/// Supervision function block - system watchdog
PROGRAM INTERNAL P_Supervision
VAR_IN_OUT
	/// Safets IOs
	stIO_Cabinet		: ST_ControlCabinetIO;
		
	/// Logger
	nLogger				: I_Logger;
END_VAR
VAR_INPUT
END_VAR
VAR_OUTPUT
	bError				: BOOL;	
	bWarning			: BOOL;
	
	bCycleStop			: BOOL;
	bFastStop			: BOOL;
END_VAR
VAR
	/// event handler
	IEvent			: I_EventHandler;
	
	/// Hardware diag FB
	fbDiagEtherCAT	: FB_DiagEtherCAT;
	
	/// private var's
	aa									: INT;	
	rTrigMachineStop_Cycle				: R_TRIG;
	rTrigMachineStop_Fast				: R_TRIG;
	tonRstStillstw						: TON;
END_VAR

/// 
/// supervision function block of the project
/// 

// reset

// run supervision (ES, Safety signals, IO-errors, etc.)

// HW diagnostics
M_EcSupervision();
M_ControlCabinet_A01();

// task cycle time exceeded
IF Statics.stPlcSystemInfo.stPlcTaskSystemInfo.CycleTimeExceeded THEN
	IEvent.Select(TC_Events.SystemEventClass.ErrorEvent)
		  .ArgSetWString(stTextListGlobal.stText_System.stText_CycletimeExceeded.wsName)
		  .Raise();	
END_IF


//-------------------------------------------------------------------------------------------------------------

IF HMI.stHmi.stIn.stMain.stButton_Start.bClick AND NOT stGlobalModuleInfo.bStation_All_Auto AND P_Safety.OpMode_Auto THEN
	IEvent.Select(TC_Events.SystemEventClass.InfoEvent)
		  .ArgSetString('Start Auto nicht moeglich -> Station nicht in Betriebsart Auto')
		  .Raise();
END_IF


//-------------------------------------------------------------------------------------------------------------

IF HMI.stHmi.stIn.stMain.stButton_Start.bClick AND NOT P_Safety.OpMode_Auto THEN
	IEvent.Select(TC_Events.SystemEventClass.InfoEvent)
		  .ArgSetString('Start Auto nicht moeglich -> Schlüsselschalter nicht auf Auto')
		  .Raise();
END_IF


//ToDo: stop / fast stop on alarm trigger
//rTrigMachineStop_Cycle(CLK := Services.fbNotiHandler.stNotificationData.eAlarmStopMode = E_EventReaction.CycleStop, Q => bCycleStop);
//rTrigMachineStop_Fast(CLK := Services.fbNotiHandler.stNotificationData.eAlarmStopMode = E_EventReaction.Stop, Q => bFastStop);

/// System error level
{attribute 'monitoring' := 'call'}
PROPERTY Error : BOOL
GET // INTERNAL
Error := bError;
END_GET
END_PROPERTY

METHOD PRIVATE M_ControlCabinet_A01 : BOOL
VAR_INPUT
END_VAR
// EC-Error
IF IO.stControlCabinetIO.stIn.IarrEcStates[E_EtherCatBox.eEtherCatBox_ControlCabinet] <> 8 THEN
	IEvent.Select(TC_Events.EtherCatEventClass.ErrorEvent)
		  .ArgSetString('EtherCatBox Control Cabinet | EC State Error')
		  .Raise();
ELSIF IO.stControlCabinetIO.stIn.IarrEcStates[E_EtherCatBox.eEtherCatBox_Oven_A] <> 8 THEN
	IEvent.Select(TC_Events.EtherCatEventClass.ErrorEvent)
		  .ArgSetString('EtherCatBox Oven A | EC State Error')
		  .Raise();
ELSIF IO.stControlCabinetIO.stIn.IarrEcStates[E_EtherCatBox.eEtherCatBox_Oven_B] <> 8 THEN
	IEvent.Select(TC_Events.EtherCatEventClass.ErrorEvent)
		  .ArgSetString('EtherCatBox Oven B | EC State Error')
		  .Raise();
ELSIF IO.stControlCabinetIO.stIn.IarrEcStates[E_EtherCatBox.eEtherCatBox_Storage] <> 8 THEN
	IEvent.Select(TC_Events.EtherCatEventClass.ErrorEvent)
		  .ArgSetString('EtherCatBox Storage | EC State Error')
		  .Raise();
END_IF
			  
(*	24V-Versorgung Netzgerät 1 Schutzschalter	
ELSIF NOT IO.stControlCabinetIO.stIn.stA01.b24V_NetzSchutz1Ok THEN
	IEvent.Select(TC_Events.HardwareEventClass.ErrorEvent)
			  .ArgSetString('=A01.G10-1QA1 | 24V-Versorgung Netzgerät 1 Schutzschalter NOK')
			  .Raise();
END_IF
*)
END_METHOD

METHOD PRIVATE M_EcSupervision : BOOL
VAR_INPUT
END_VAR
VAR_INST

END_VAR

// automatic EC supervision
fbDiagEtherCAT();

(*
//IarrEcState
// Diag EC Boxes for fast reaction				
IF (stIO_Cabinet.stIn.IarrEcStates[1] <> 8) THEN
	bError:=TRUE;
	fbNotiHandler.M_SetNotificationEx(F_CreateDynText("403",403),
									stTextListGlobal.stText_NG_Hardware, 
									stTextListGlobal.stText_EtherCatBox_Error, "++M1+E2-57CO1 (CU1128)", stTextListGlobal.stText_EtherCatBox_OP_Error, 
									E_AlarmPriority.Error, E_NotificationMode.eNotificationMode_Reset);	
END_IF
IF (stIO_Cabinet.stIn.IarrEcStates[2] <> 8) THEN
	bError:=TRUE;
	fbNotiHandler.M_SetNotificationEx(F_CreateDynText("404",404),
									stTextListGlobal.stText_NG_Hardware, 
									stTextListGlobal.stText_EtherCatBox_Error, "++M1+E2-57CO1 (CU1128-B)", stTextListGlobal.stText_EtherCatBox_OP_Error, 
									E_AlarmPriority.Error, E_NotificationMode.eNotificationMode_Reset);	
END_IF
IF (stIO_Cabinet.stIn.IarrEcStates[3] <> 8) THEN
	bError:=TRUE;
	fbNotiHandler.M_SetNotificationEx(F_CreateDynText("405",405),
									stTextListGlobal.stText_NG_Hardware, 
									stTextListGlobal.stText_EtherCatBox_Error, "++M1+E2-57CO1 (CU1128-C)", stTextListGlobal.stText_EtherCatBox_OP_Error, 
									E_AlarmPriority.Error, E_NotificationMode.eNotificationMode_Reset);	
END_IF
IF (stIO_Cabinet.stIn.IarrEcStates[4] <> 8) THEN
	bError:=TRUE;
	fbNotiHandler.M_SetNotificationEx(F_CreateDynText("406",406),
									stTextListGlobal.stText_NG_Hardware, 
									stTextListGlobal.stText_EtherCatBox_Error, "++M1+E2-62BC1 (EK1100)", stTextListGlobal.stText_EtherCatBox_OP_Error, 
									E_AlarmPriority.Error, E_NotificationMode.eNotificationMode_Reset);	
END_IF
IF (stIO_Cabinet.stIn.IarrEcStates[5] <> 8) THEN
	bError:=TRUE;
	fbNotiHandler.M_SetNotificationEx(F_CreateDynText("407",407),
									stTextListGlobal.stText_NG_Hardware, 
									stTextListGlobal.stText_EtherCatBox_Error, "++A1+P1-4A2 (EP2338-0002)", stTextListGlobal.stText_EtherCatBox_OP_Error, 
									E_AlarmPriority.Error, E_NotificationMode.eNotificationMode_Reset);	
END_IF
IF (stIO_Cabinet.stIn.IarrEcStates[6] <> 8) THEN
	bError:=TRUE;
	fbNotiHandler.M_SetNotificationEx(F_CreateDynText("0",0),
									stTextListGlobal.stText_NG_Hardware, 
									stTextListGlobal.stText_EtherCatBox_Error, "++A1+P1-5SI0 (EP1908)", stTextListGlobal.stText_EtherCatBox_OP_Error, 
									E_AlarmPriority.Error, E_NotificationMode.eNotificationMode_Reset);	
END_IF
IF (stIO_Cabinet.stIn.IarrEcStates[7] <> 8)  THEN
	bError:=TRUE;
	fbNotiHandler.M_SetNotificationEx(F_CreateDynText("408",408),
									stTextListGlobal.stText_NG_Hardware, 
									stTextListGlobal.stText_EtherCatBox_Error, "++A1+P1-6SI0 (EP1908)", stTextListGlobal.stText_EtherCatBox_OP_Error, 
									E_AlarmPriority.Error, E_NotificationMode.eNotificationMode_Reset);	
END_IF
IF (stIO_Cabinet.stIn.IarrEcStates[8] <> 8) THEN
	bError:=TRUE;
	fbNotiHandler.M_SetNotificationEx(F_CreateDynText("409",409),
									stTextListGlobal.stText_NG_Hardware, 
									stTextListGlobal.stText_EtherCatBox_Error, "++A1+P1-3A2 (EP2338-0002)", stTextListGlobal.stText_EtherCatBox_OP_Error, 
									E_AlarmPriority.Error, E_NotificationMode.eNotificationMode_Reset);	
END_IF

IF (stIO_Cabinet.stIn.IarrEcStates[9] <> 8) THEN
	bError:=TRUE;
	fbNotiHandler.M_SetNotificationEx(F_CreateDynText("410",410),
									stTextListGlobal.stText_NG_Hardware, 
									stTextListGlobal.stText_EtherCatBox_Error, "++M1+E1-46BC3 (EK1100)", stTextListGlobal.stText_EtherCatBox_OP_Error, 
									E_AlarmPriority.Error, E_NotificationMode.eNotificationMode_Reset);	
END_IF
IF (stIO_Cabinet.stIn.IarrEcStates[10] <> 8) THEN
	bError:=TRUE;
	fbNotiHandler.M_SetNotificationEx(F_CreateDynText("411",411),
									stTextListGlobal.stText_NG_Hardware, 
									stTextListGlobal.stText_EtherCatBox_Error, "++M1+E1-38U1 (AX5206-0000-0213)", stTextListGlobal.stText_EtherCatBox_OP_Error, 
									E_AlarmPriority.Error, E_NotificationMode.eNotificationMode_Reset);	
END_IF
IF (stIO_Cabinet.stIn.IarrEcStates[11] <> 8) THEN
	bError:=TRUE;
	fbNotiHandler.M_SetNotificationEx(F_CreateDynText("412",412),
									stTextListGlobal.stText_NG_Hardware, 
									stTextListGlobal.stText_EtherCatBox_Error, "++M1+E1-31U1 (Rtt)", stTextListGlobal.stText_EtherCatBox_OP_Error, 
									E_AlarmPriority.Error, E_NotificationMode.eNotificationMode_Reset);	
END_IF
IF (stIO_Cabinet.stIn.IarrEcStates[12] <> 8) THEN
	bError:=TRUE;
	fbNotiHandler.M_SetNotificationEx(F_CreateDynText("413",413),
									stTextListGlobal.stText_NG_Hardware, 
									stTextListGlobal.stText_EtherCatBox_Error, "++M1+Festo_V1 (CPX-FB37)", stTextListGlobal.stText_EtherCatBox_OP_Error, 
									E_AlarmPriority.Error, E_NotificationMode.eNotificationMode_Reset);	
END_IF
IF (stIO_Cabinet.stIn.IarrEcStates[13] <> 8) THEN
	bError:=TRUE;
	fbNotiHandler.M_SetNotificationEx(F_CreateDynText("414",414),
									stTextListGlobal.stText_NG_Hardware, 
									stTextListGlobal.stText_EtherCatBox_Error, "++M1+KeyenceSR_X100-30U1 (SR-EC1)", stTextListGlobal.stText_EtherCatBox_OP_Error, 
									E_AlarmPriority.Error, E_NotificationMode.eNotificationMode_Reset);	
END_IF
*)
END_METHOD

METHOD INTERNAL M_Init : BOOL
VAR_INPUT
END_VAR
SetReferences(Services.fbEventHandler);
END_METHOD

/// resets all notification flags and reset-needed state 
METHOD M_Reset
VAR
	ii: INT;
END_VAR
// reset error level
nLogger.AddLog(Concat2x('Reset, Error: ', TO_STRING(bError)), 'Supervision', eLogLevel_info);
bError := FALSE;
bWarning := FALSE;
END_METHOD

/// Dependency injection method.
{attribute 'object_name' := 'SetReferences'}
METHOD INTERNAL SetReferences
VAR_INPUT
	/// event access provider
	IEventHandler : I_EventHandler;
END_VAR
// init components stuff here...
IEvent := IEventHandler;
fbDiagEtherCAT.SetReferences(IEvent);
END_METHOD

END_PROGRAM

(* stored: Version 1.1.0.1
   POU P_Supervision: Id {27b53e36-c41d-419b-b0d2-7542c866bd49}, SpecialFunc None
   Folder ControlCabinets: Id {3b83c655-d8bd-4570-b761-65c2f46173a3}
   Folder EtherCat: Id {e6ad6cad-7361-43c9-ae82-fc5a632fa144}
   Folder Properties: Id {e6c31f63-b52a-4b3c-898a-95bec3af0620}
   Property Error: Id {3e5ee790-8a5a-4345-9130-0b2d747e0157}
   Get Get: Id {85cc22c1-ab63-4cc1-b1c8-d9fd0fbdb774}
   Method M_ControlCabinet_A01: Id {f75c048d-9e5b-4543-8b0a-6132207d9d8b}
   Method M_EcSupervision: Id {a1825d9d-758b-4143-bce6-ae5a64f5cc86}
   Method M_Init: Id {6c1e11de-3f73-4bf5-9c70-38c4750f8404}
   Method M_Reset: Id {4862ee2f-425b-44b5-bbdb-f1e78a7f4da0}
   Method SetReferences: Id {3b378dd0-c1c9-4636-9d61-e83ef672d4ac} *)
